// Mitsubishi GX Works2 project: 서보컨베이어제어   PLC: Q03UD

PROGRAM MAIN
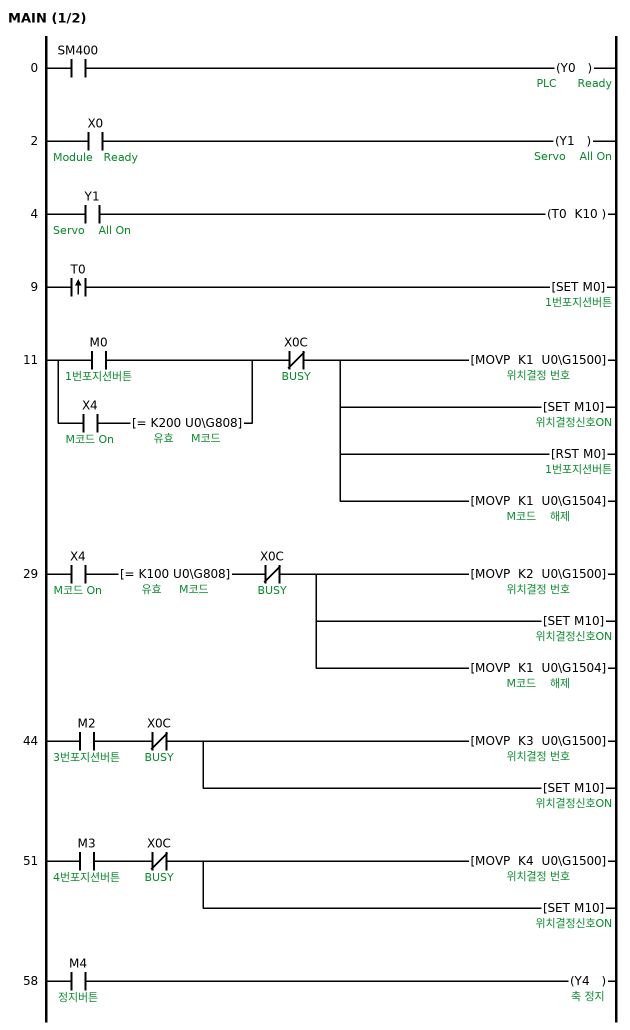
0     LD      SM400
      OUT     Y0  ; PLC      Ready
2     LD      X0  ; Module   Ready
      OUT     Y1  ; Servo    All On
4     LD      Y1  ; Servo    All On
      OUT     T0 K10
9     LDP     T0
      SET     M0  ; 1번포지션버튼
11    LD      M0  ; 1번포지션버튼
      LD      X4  ; M코드 On
      AND=    K200 U0\G808  ; 유효     M코드
      ORB
      ANI     X0C  ; BUSY
      MOVP    K1 U0\G1500  ; 위치결정 번호
      SET     M10  ; 위치결정신호ON
      RST     M0  ; 1번포지션버튼
      MOVP    K1 U0\G1504  ; M코드    해제
29    LD      X4  ; M코드 On
      AND=    K100 U0\G808  ; 유효     M코드
      ANI     X0C  ; BUSY
      MOVP    K2 U0\G1500
      SET     M10  ; 위치결정신호ON
      MOVP    K1 U0\G1504
44    LD      M2  ; 3번포지션버튼
      ANI     X0C  ; BUSY
      MOVP    K3 U0\G1500
      SET     M10  ; 위치결정신호ON
51    LD      M3  ; 4번포지션버튼
      ANI     X0C  ; BUSY
      MOVP    K4 U0\G1500
      SET     M10  ; 위치결정신호ON
58    LD      M4  ; 정지버튼
      OUT     Y4  ; 축 정지
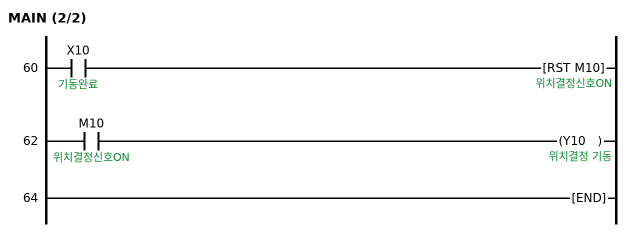
60    LD      X10  ; 기동완료
      RST     M10  ; 위치결정신호ON
62    LD      M10  ; 위치결정신호ON
      OUT     Y10  ; 위치결정 기동
64    END
END_PROGRAM

// device comments not shown above
X14  ; 위치결정 완료
M1  ; 2번포지션버튼
